FUNCTION_BLOCK _SEPARATE EXTENDS FB_STATION
VAR_INPUT
	b_BULL_SENSOR:BOOL:=FALSE;
	piston_updown: REFERENCE TO FB_PIST;
	piston_colet1: REFERENCE TO FB_PIST;
	piston_colet2: REFERENCE TO FB_PIST;
	piston_colet3: REFERENCE TO FB_PIST;
	piston_colet4: REFERENCE TO FB_PIST;
	piston_puller: REFERENCE TO FB_PIST;
	piston_tray: REFERENCE TO FB_PIST;
	piston_pins: REFERENCE TO FB_PIST;
	piston_tray_door: REFERENCE TO FB_PIST;
	piston_tray_push: REFERENCE TO FB_PIST;
	bInit:BOOL:=FALSE;
	
	
	fbAxis:REFERENCE TO FB_Axis;
	
END_VAR
VAR_OUTPUT
	bRUNNING:BOOL :=FALSE;
	bError:BOOL:=FALSE;
END_VAR
VAR
	//bHomed:BOOL :=FALSE;
	tDelay: TON;
	bDELAY: BOOL:=FALSE;
	E: INT;
	
	//bDone: BOOL;
	step_timeout: TIME:=T#7S;
	colet_close: INT;
END_VAR


act();

CASE eState OF
	
	E_STATION_STATE.homing:
		//SFCReset:=FALSE;
		//SFCInit:=FALSE;
		piston_updown.A_INIT();
		piston_colet1.A_INIT(); piston_colet2.A_INIT();piston_colet3.A_INIT();piston_colet4.A_INIT();
		piston_tray.A_INIT();
		piston_tray_push.A_INIT();
		piston_tray_door.A_INIT();
		piston_pins.A_INIT();
		eState:= E_STATION_STATE.idle;
		bHomed:=TRUE;
		bError:=FALSE;
		//axis-------------------
		fbAxis.bEnable:=TRUE;
		fbAxis.bHalt:=FALSE;
		fbAxis.bSetPosition:=FALSE;
		fbAxis.bReset:=FALSE;
		
	E_STATION_STATE.uninit:
		eState:= E_STATION_STATE.homing;
		fbAxis.bDo_Step_FW:=FALSE;
		fbAxis.bMoveRel:=FALSE;
		fbAxis.stepFW_state:=0;
		fbAxis.bHalt:=FALSE;
		fbAxis.bReset:=FALSE;

	E_STATION_STATE.idle:
		//idle
		
	E_STATION_STATE.do_action1://delay and lower device
		//main action
		
	E_STATION_STATE.done:
		//dd
	 
	E_STATION_STATE.pause:
		//paused
	
	E_STATION_STATE.error:
		//error
	
	E_STATION_STATE.estop:
		fbAxis.stepFW_state:=0;
		fbAxis.bHalt:=TRUE;
		fbAxis.bReset:=TRUE;
		bHomed:=FALSE;

END_CASE

ACTION _aCLOSE_COLET_1_4_active:
IF  NOT (eState = E_STATION_STATE.pause) THEN
bDone:=TRUE;
END_IF
END_ACTION

ACTION _aCLOSE_COLET_1_4_entry:

	bDone:=FALSE;
	IF NOT (eState = E_STATION_STATE.pause) THEN
		piston_colet1.A_OPEN();
		piston_colet4.A_OPEN();
		piston_pins.A_OPEN();
		
	END_IF
END_ACTION

ACTION _aCLOSE_COLET_active:
IF NOT (eState = E_STATION_STATE.pause) THEN

//IF piston_colet1.pistStatus= E_PIST_STATUS.OPENED AND piston_colet2.pistStatus= E_PIST_STATUS.OPENED THEN
	bDone:=TRUE;
//END_IF

END_IF
END_ACTION

ACTION _aCLOSE_COLET_entry:

	bDone:=FALSE;
	IF NOT (eState = E_STATION_STATE.pause) THEN
		piston_colet2.A_OPEN();
		piston_colet3.A_OPEN();
		
	END_IF
END_ACTION

ACTION _aIDLE_active:
IF eState = E_STATION_STATE.do_action1 THEN 
	bDone:=TRUE;
	
END_IF
END_ACTION

ACTION _aIDLE_entry:
bDone:=FALSE;
END_ACTION

ACTION _aJACK_UP1_active:
IF JACK_UP1.t>step_timeout AND NOT (eState = E_STATION_STATE.pause)THEN
		bERROR:=TRUE;
END_IF
IF fbAxis.RELATIVE.Done THEN
	bDone:=TRUE;
END_IF
END_ACTION

ACTION _aJACK_UP1_entry:

	bDone:=FALSE;
	IF NOT (eState = E_STATION_STATE.pause) THEN
		piston_updown.A_NEUTRAL();
		fbAxis.bDo_Step_FW:=TRUE;
		
	END_IF
END_ACTION

ACTION _aJACK_UP2_active:
IF JACK_UP2.t>step_timeout AND NOT (eState = E_STATION_STATE.pause) THEN
		bERROR:=TRUE;
END_IF
IF fbAxis.RELATIVE.Done THEN
	bDone:=TRUE;
END_IF
END_ACTION

ACTION _aJACK_UP2_entry:

	bDone:=FALSE;
	IF NOT (eState = E_STATION_STATE.pause) THEN
		fbAxis.bDo_Step_FW:=TRUE;
		
	END_IF
END_ACTION

ACTION _aLOWER_LIFT_active:
IF LOWER_LIFT.t>step_timeout AND NOT (eState = E_STATION_STATE.pause) THEN
		bERROR:=TRUE;
END_IF

IF piston_updown.pistStatus= E_PIST_STATUS.OPENED   THEN
	bDone:=TRUE;
END_IF
END_ACTION

ACTION _aLOWER_LIFT_entry:

	bDone:=FALSE;
	IF NOT bSkip AND NOT (eState = E_STATION_STATE.pause) THEN
		piston_updown.A_OPEN();	
		
	ELSE
		eState:=E_STATION_STATE.done;
	END_IF
END_ACTION

ACTION _aOPEN_COLETS_active:
IF OPEN_COLETS.t>step_timeout AND NOT (eState = E_STATION_STATE.pause) THEN
		bERROR:=TRUE;
END_IF

IF piston_colet1.pistStatus= E_PIST_STATUS.CLOSED AND piston_colet2.pistStatus= E_PIST_STATUS.CLOSED AND piston_colet3.pistStatus= E_PIST_STATUS.CLOSED AND piston_colet4.pistStatus= E_PIST_STATUS.CLOSED THEN
	bDone:=TRUE;
END_IF
END_ACTION

ACTION _aOPEN_COLETS_entry:

	bDone:=FALSE;
	IF NOT (eState = E_STATION_STATE.pause) THEN
		piston_colet2.A_CLOSE();
		piston_colet3.A_CLOSE();
		piston_colet1.A_CLOSE();
		piston_colet4.A_CLOSE();
		
	END_IF
END_ACTION

ACTION _aPINS_DOWN_active:
IF PINS_DOWN.t>step_timeout AND NOT (eState = E_STATION_STATE.pause) THEN
		bERROR:=TRUE;
END_IF

IF piston_pins.pistStatus= E_PIST_STATUS.OPENED THEN
	bDone:=TRUE;
END_IF
END_ACTION

ACTION _aPINS_DOWN_entry:

	bDone:=FALSE;
	IF NOT (eState = E_STATION_STATE.pause) THEN
		piston_pins.A_OPEN();
	END_IF
END_ACTION

ACTION _aPINS_UP_active:
IF PINS_UP.t>step_timeout AND NOT (eState = E_STATION_STATE.pause) THEN
		bERROR:=TRUE;
END_IF

IF piston_pins.pistStatus= E_PIST_STATUS.CLOSED THEN
	bDone:=TRUE;
END_IF
END_ACTION

ACTION _aPINS_UP_entry:

	bDone:=FALSE;
	IF NOT (eState = E_STATION_STATE.pause) THEN
		piston_pins.A_CLOSE();
	END_IF
END_ACTION

ACTION _aRAISE_LIFT_active:
IF RAISE_LIFT.t>step_timeout AND NOT (eState = E_STATION_STATE.pause) THEN
		bERROR:=TRUE;
END_IF

IF piston_updown.pistStatus= E_PIST_STATUS.CLOSED THEN
	bDone:=TRUE;
END_IF
END_ACTION

ACTION _aRAISE_LIFT_entry:

	bDone:=FALSE;
	IF NOT (eState = E_STATION_STATE.pause) THEN
		piston_updown.A_CLOSE();
	END_IF
END_ACTION

ACTION _aTRAY_active:
IF TRAY.t>step_timeout AND NOT (eState = E_STATION_STATE.pause) THEN
		bERROR:=TRUE;
END_IF

IF piston_tray.pistStatus= E_PIST_STATUS.OPENED THEN
	bDone:=TRUE;
END_IF
END_ACTION

ACTION _aTRAY_entry:

	bDone:=FALSE;
	IF NOT (eState = E_STATION_STATE.pause) THEN
		piston_tray.A_OPEN();
	END_IF
END_ACTION

ACTION _aTRAY_JACK_BACK_active:
IF NOT (eState = E_STATION_STATE.pause) THEN
	eState:= E_STATION_STATE.done;
	bDone:=TRUE;
END_IF
END_ACTION

ACTION _aUNINIT_entry:
bDone:=TRUE;
END_ACTION

ACTION act:
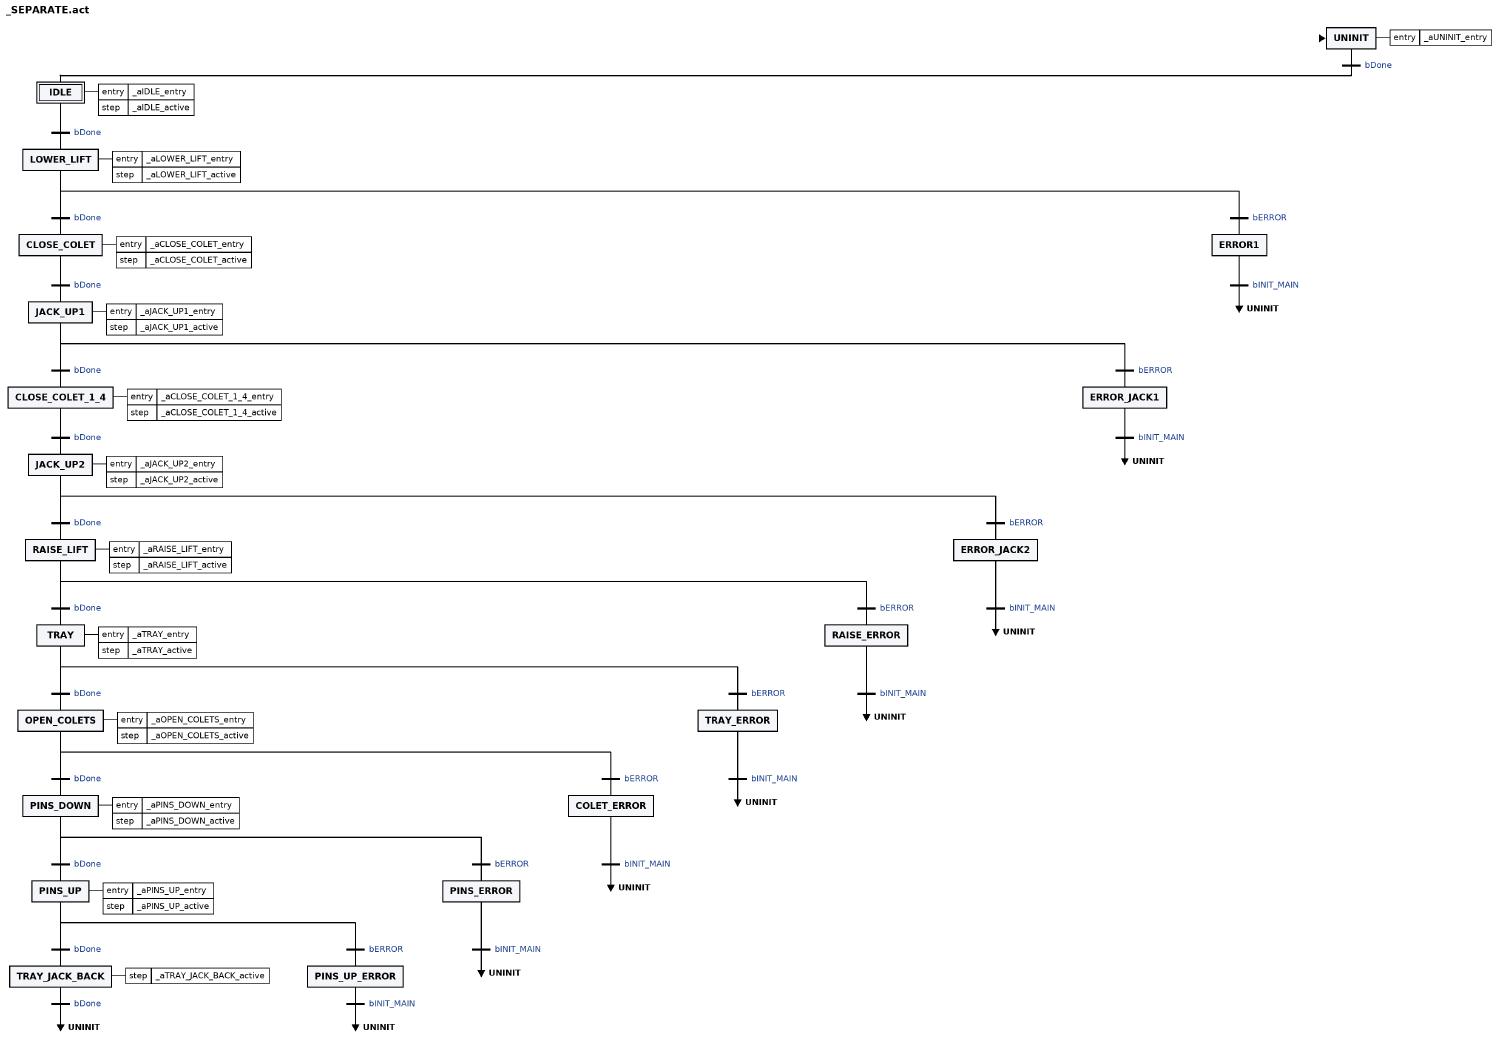
STEP UNINIT:
    _aUNINIT_entry(P1);  // entry action
END_STEP
TRANSITION FROM UNINIT TO IDLE
    := bDone;
END_TRANSITION
INITIAL_STEP IDLE:
    _aIDLE_entry(P1);  // entry action
    _aIDLE_active(N);  // step action
END_STEP
TRANSITION FROM IDLE TO LOWER_LIFT
    := bDone;
END_TRANSITION
STEP LOWER_LIFT:
    _aLOWER_LIFT_entry(P1);  // entry action
    _aLOWER_LIFT_active(N);  // step action
END_STEP
TRANSITION FROM LOWER_LIFT TO CLOSE_COLET
    := bDone;
END_TRANSITION
STEP CLOSE_COLET:  // min time T#1s
    _aCLOSE_COLET_entry(P1);  // entry action
    _aCLOSE_COLET_active(N);  // step action
END_STEP
TRANSITION FROM CLOSE_COLET TO JACK_UP1
    := bDone;
END_TRANSITION
STEP JACK_UP1:  // min time T#2s
    _aJACK_UP1_entry(P1);  // entry action
    _aJACK_UP1_active(N);  // step action
END_STEP
TRANSITION FROM JACK_UP1 TO CLOSE_COLET_1_4
    := bDone;
END_TRANSITION
STEP CLOSE_COLET_1_4:
    _aCLOSE_COLET_1_4_entry(P1);  // entry action
    _aCLOSE_COLET_1_4_active(N);  // step action
END_STEP
TRANSITION FROM CLOSE_COLET_1_4 TO JACK_UP2
    := bDone;
END_TRANSITION
STEP JACK_UP2:  // min time T#2s
    _aJACK_UP2_entry(P1);  // entry action
    _aJACK_UP2_active(N);  // step action
END_STEP
TRANSITION FROM JACK_UP2 TO RAISE_LIFT
    := bDone;
END_TRANSITION
STEP RAISE_LIFT:
    _aRAISE_LIFT_entry(P1);  // entry action
    _aRAISE_LIFT_active(N);  // step action
END_STEP
TRANSITION FROM RAISE_LIFT TO TRAY
    := bDone;
END_TRANSITION
STEP TRAY:
    _aTRAY_entry(P1);  // entry action
    _aTRAY_active(N);  // step action
END_STEP
TRANSITION FROM TRAY TO OPEN_COLETS
    := bDone;
END_TRANSITION
STEP OPEN_COLETS:
    _aOPEN_COLETS_entry(P1);  // entry action
    _aOPEN_COLETS_active(N);  // step action
END_STEP
TRANSITION FROM OPEN_COLETS TO PINS_DOWN
    := bDone;
END_TRANSITION
TRANSITION FROM OPEN_COLETS TO COLET_ERROR
    := bERROR;
END_TRANSITION
STEP COLET_ERROR:
END_STEP
TRANSITION FROM COLET_ERROR TO UNINIT
    := bINIT_MAIN;
END_TRANSITION
STEP PINS_DOWN:
    _aPINS_DOWN_entry(P1);  // entry action
    _aPINS_DOWN_active(N);  // step action
END_STEP
TRANSITION FROM PINS_DOWN TO PINS_UP
    := bDone;
END_TRANSITION
STEP PINS_UP:
    _aPINS_UP_entry(P1);  // entry action
    _aPINS_UP_active(N);  // step action
END_STEP
TRANSITION FROM PINS_UP TO TRAY_JACK_BACK
    := bDone;
END_TRANSITION
STEP TRAY_JACK_BACK:
    _aTRAY_JACK_BACK_active(N);  // step action
END_STEP
TRANSITION FROM TRAY_JACK_BACK TO UNINIT
    := bDone;
END_TRANSITION
TRANSITION FROM PINS_UP TO PINS_UP_ERROR
    := bERROR;
END_TRANSITION
STEP PINS_UP_ERROR:
END_STEP
TRANSITION FROM PINS_UP_ERROR TO UNINIT
    := bINIT_MAIN;
END_TRANSITION
TRANSITION FROM PINS_DOWN TO PINS_ERROR
    := bERROR;
END_TRANSITION
STEP PINS_ERROR:
END_STEP
TRANSITION FROM PINS_ERROR TO UNINIT
    := bINIT_MAIN;
END_TRANSITION
TRANSITION FROM TRAY TO TRAY_ERROR
    := bERROR;
END_TRANSITION
STEP TRAY_ERROR:
END_STEP
TRANSITION FROM TRAY_ERROR TO UNINIT
    := bINIT_MAIN;
END_TRANSITION
TRANSITION FROM RAISE_LIFT TO RAISE_ERROR
    := bERROR;
END_TRANSITION
STEP RAISE_ERROR:
END_STEP
TRANSITION FROM RAISE_ERROR TO UNINIT
    := bINIT_MAIN;
END_TRANSITION
TRANSITION FROM JACK_UP2 TO ERROR_JACK2
    := bERROR;
END_TRANSITION
STEP ERROR_JACK2:
END_STEP
TRANSITION FROM ERROR_JACK2 TO UNINIT
    := bINIT_MAIN;
END_TRANSITION
TRANSITION FROM JACK_UP1 TO ERROR_JACK1
    := bERROR;
END_TRANSITION
STEP ERROR_JACK1:
END_STEP
TRANSITION FROM ERROR_JACK1 TO UNINIT
    := bINIT_MAIN;
END_TRANSITION
TRANSITION FROM LOWER_LIFT TO ERROR1
    := bERROR;
END_TRANSITION
STEP ERROR1:
END_STEP
TRANSITION FROM ERROR1 TO UNINIT
    := bINIT_MAIN;
END_TRANSITION
// branch label Branch7_act
// branch label Branch8_act
// branch label Branch6_act
// branch label Branch5_act
// branch label Branch4_act
// branch label Branch3_act
// branch label Branch2_act
// branch label Branch0_act
END_ACTION

END_FUNCTION_BLOCK

(* stored: Version 1.1.0.1, ProductVersion 3.1.4024.12
   POU _SEPARATE: Id {774d5f23-7f9c-4716-a2b6-be8a6039a8a9}, SpecialFunc None
   Folder ACT: Id {85bdc405-ef8a-4ef0-bec7-0df14e5fed51}
   Action _aCLOSE_COLET_1_4_active: Id {04875a07-6118-4ff1-8c19-c49e1593d52a}
   Action _aCLOSE_COLET_1_4_entry: Id {f0d544cd-22bf-4975-bb02-e00bc67879c5}
   Action _aCLOSE_COLET_active: Id {973f3047-ddb6-495b-bc23-4e92976e27ee}
   Action _aCLOSE_COLET_entry: Id {3a15b879-37b5-48be-bd24-8c84beec22df}
   Action _aIDLE_active: Id {af40f943-e48b-4482-bb18-e5fb59e1ef74}
   Action _aIDLE_entry: Id {517c51b4-0342-4521-a997-9b2976ea4d7b}
   Action _aJACK_UP1_active: Id {9ff3f380-dce0-4cbf-b2bd-4b2cd0955ccc}
   Action _aJACK_UP1_entry: Id {e2ff9f94-709e-49ce-9afa-1abc1b23db96}
   Action _aJACK_UP2_active: Id {5fa746e2-bbe2-4608-b163-e36a11e222b8}
   Action _aJACK_UP2_entry: Id {45a0ca18-f995-4302-ba88-4c25db84b817}
   Action _aLOWER_LIFT_active: Id {1c5f6484-78e2-4838-8619-33c6be408816}
   Action _aLOWER_LIFT_entry: Id {81f257de-9e43-4a8c-997a-59be3c9b9359}
   Action _aOPEN_COLETS_active: Id {37f536be-af98-413b-8869-c66286beaae5}
   Action _aOPEN_COLETS_entry: Id {ca5e7a84-cd7d-4cc6-9d57-6be88a5d0e94}
   Action _aPINS_DOWN_active: Id {5ae94f0d-bd82-4f9f-bce9-77ae8546598d}
   Action _aPINS_DOWN_entry: Id {086fff13-3831-48fc-81c7-883890abed30}
   Action _aPINS_UP_active: Id {182c0292-75a2-4eb5-a792-3bd9fec3f93e}
   Action _aPINS_UP_entry: Id {01423d15-a6ae-45b9-8427-f2babbaf4eb7}
   Action _aRAISE_LIFT_active: Id {f781ea8a-d611-41fa-bf36-752be68f618f}
   Action _aRAISE_LIFT_entry: Id {c0715746-6732-43ef-96ea-ec4f55ac6c85}
   Action _aTRAY_active: Id {16938058-a5c2-46c8-81e5-edb1e59082fc}
   Action _aTRAY_entry: Id {e1b1d132-5545-478a-8894-bd1a2ee594ba}
   Action _aTRAY_JACK_BACK_active: Id {ec1ead27-56b8-4560-959a-ffdb827fb9c7}
   Action _aUNINIT_entry: Id {3524b8ee-e3dc-4082-b5dd-f8d85280042e}
   Action act: Id {2f3a4461-d0bc-40c6-bcdf-e8b08b6b9f73} *)
